Yaskawa INFORM job: TWIN_FRONT_WELD_-90ST-2_5340.JBI

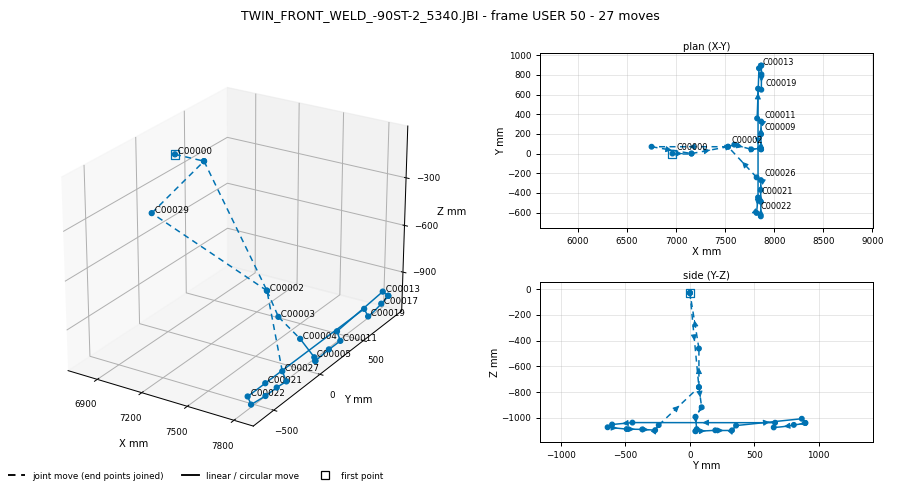
[picture p0: tool path of TWIN_FRONT_WELD_-90ST-2_5340.JBI in frame USER 50, 27 of 31 moves have a stored position in this frame; points joined in program order, loops and branches not executed]
/JOB
//NAME TWIN_FRONT_WELD_-90ST-2_5340
///FOLDERNAME 02-SKRZYNIE_JOBS
//POS
///NPOS 31,31,0,6,0,0
///USER 50
///TOOL 0
///POSTYPE USER
///RECTAN
///RCONF 0,0,1,0,0,0,0,0,0,0,0,0,0,0,0,0,0,0,0,0,0,0,0,0
C00000=6964.103,0.312,-30.113,0.0036,-53.6521,-0.0034
C00001=7158.107,0.312,-30.113,0.0036,-53.6521,-0.0034
///RCONF 1,0,0,0,0,0,0,0,0,0,0,0,0,0,0,0,0,0,0,0,0,0,0,0
C00002=7529.895,69.936,-761.128,0.1694,36.7808,-161.6994
C00003=7593.803,91.186,-917.296,-9.7230,35.0705,-163.2693
C00004=7765.973,43.237,-990.708,2.4332,41.3600,-160.2788
C00005=7854.092,52.836,-1087.295,2.4326,41.3464,-160.2685
C00006=7866.086,43.569,-1103.074,2.4250,41.3408,-160.2847
C00007=7866.672,43.652,-1103.070,2.4247,41.3414,-160.2846
C00008=7865.168,101.752,-1101.058,2.4312,41.5896,-160.2966
///RCONF 0,0,0,0,0,0,0,0,0,0,0,0,0,0,0,0,0,0,0,0,0,0,0,0
C00009=7865.744,197.178,-1096.159,2.5302,41.7008,-160.1737
C00010=7865.567,255.531,-1097.573,2.5319,41.6997,-160.1630
C00011=7866.686,326.732,-1096.309,2.5308,41.6996,-160.1597
C00012=7825.961,358.355,-1059.396,2.5279,41.7009,-160.1704
C00013=7844.512,868.318,-1006.408,-36.5717,33.3380,158.1479
C00014=7867.707,896.307,-1038.748,-33.3426,31.0834,153.4598
C00015=7867.746,895.180,-1038.953,-33.3375,31.0829,153.4546
C00016=7869.178,857.917,-1047.022,-33.1867,30.9856,153.2302
C00017=7869.794,806.472,-1054.108,-32.5616,29.0872,131.6988
C00018=7869.506,734.683,-1066.166,-32.5472,29.0702,136.7150
C00019=7868.451,650.382,-1073.764,-32.5333,29.0523,142.4520
C00020=7835.214,661.117,-1037.227,-32.5695,29.0775,153.4943
C00021=7835.222,-446.023,-1036.229,41.9938,34.9165,-143.3319
C00022=7820.199,-603.860,-1051.032,41.9928,34.9182,-143.3350
C00023=7863.342,-638.725,-1072.644,41.9898,34.9141,-143.3376
///RCONF 0,0,0,0,1,0,0,0,0,0,0,0,0,0,0,0,0,0,0,0,0,0,0,0
C00024=7863.688,-490.448,-1086.753,35.6266,29.1231,-116.2046
///RCONF 0,0,0,0,0,0,0,0,0,0,0,0,0,0,0,0,0,0,0,0,0,0,0,0
C00025=7862.301,-369.694,-1089.170,35.5308,29.0998,-115.5093
C00026=7864.181,-269.690,-1094.936,35.4517,29.0825,-114.8963
C00027=7820.806,-242.024,-1055.912,35.4344,29.0737,-114.7919
///RCONF 1,0,0,0,0,0,0,0,0,0,0,0,0,0,0,0,0,0,0,0,0,0,0,0
C00028=7529.895,69.936,-761.128,0.1694,36.7808,-161.6994
///RCONF 1,0,1,0,0,0,0,0,0,0,0,0,0,0,0,0,0,0,0,0,0,0,0,0
C00029=6751.458,69.938,-461.595,1.9967,40.9431,-160.5509
///RCONF 0,0,1,0,0,0,0,0,0,0,0,0,0,0,0,0,0,0,0,0,0,0,0,0
C00030=7158.107,0.312,-30.113,0.0036,-53.6521,-0.0034
///RCONF 0,0,0,0,0,0,0,0,0,0,0,0,0,0,0,0,0,0,0,0,0,0,0,0
BC00000=5149.685
BC00001=5343.689
BC00002=6178.800
BC00003=6423.804
BC00004=6624.475
BC00005=6624.475
BC00006=6624.495
BC00007=6624.495
BC00008=6624.488
BC00009=6624.482
BC00010=6624.482
BC00011=6624.482
BC00012=6624.482
BC00013=6624.488
BC00014=6624.488
BC00015=6624.488
BC00016=6624.476
BC00017=6624.489
BC00018=6624.489
BC00019=6624.228
BC00020=6624.488
BC00021=6624.488
BC00022=6624.482
BC00023=6624.482
BC00024=6624.469
BC00025=6624.475
BC00026=6624.482
BC00027=6624.482
BC00028=6178.800
BC00029=5343.689
BC00030=5343.689
///POSTYPE BASE
///RCONF 1,0,0,0,0,0,0,0,0,0,0,0,0,0,0,0,0,0,0,0,0,0,0,0
P00500=2.332,-5.281,-1.258,0.0000,0.0000,0.0000
///RCONF 0,0,0,0,0,0,0,0,0,0,0,0,0,0,0,0,0,0,0,0,0,0,0,0
P00501=-2.026,0.009,3.534,0.0000,0.0000,0.0000
///RCONF 1,0,0,0,0,0,0,0,0,0,0,0,0,0,0,0,0,0,0,0,0,0,0,0
P00502=-2.023,0.001,1.732,0.0000,0.0000,0.0000
P00503=0.138,-0.044,1.539,0.0000,0.0000,0.0000
P00504=-0.309,-0.010,1.636,0.0000,0.0000,0.0000
P00505=0.999,-9.916,8.214,0.0000,0.0000,0.0000
//INST
///DATE 2024/12/18 15:54
///ATTR SC,RW,RJ
////FRAME USER 50
///GROUP1 RB1,BS1
NOP
MOVJ C00000 BC00000 VJ=60.00
MOVJ C00001 BC00001 VJ=60.00
MOVJ C00002 BC00002 VJ=60.00
MOVJ C00003 BC00003 VJ=60.00
MOVJ C00004 BC00004 VJ=30.00
'::::::::::::::::::::::::::::::::
'W20
'::::::::::::::::::::::::::::::::
MOVL C00005 BC00005 V=333.3
SFTON P0503
MACRO1 MJ#(0) ARGF14
MOVL C00006 BC00006 V=166.7 PL=0
ARCON
MOVC C00007 BC00007 V=9.5
MOVC C00008 BC00008 V=9.5
MOVC C00009 BC00009 V=9.5
SFTOF
SFTON P0502
MOVC C00010 BC00010 V=9.5
MOVC C00011 BC00011 V=9.5
ARCOF
MOVL C00012 BC00012 V=166.7
SFTOF
'::::::::::::::::::::::::::::::::
'W21
'::::::::::::::::::::::::::::::::
MOVL C00013 BC00013 V=333.3
SFTON P0500
MACRO1 MJ#(0) ARGF14
MOVL C00014 BC00014 V=166.7 PL=0
ARCON
MOVC C00015 BC00015 V=9.5
MOVC C00016 BC00016 V=9.5
MOVC C00017 BC00017 V=9.5
SFTOF
SFTON P0501
MOVC C00018 BC00018 V=9.5
MOVC C00019 BC00019 V=9.5
ARCOF
MOVL C00020 BC00020 V=166.7
SFTOF
MOVL C00021 BC00021 V=333.3
'::::::::::::::::::::::::::::::::
'W22
'::::::::::::::::::::::::::::::::
MOVL C00022 BC00022 V=333.3
SFTON P0505
MACRO1 MJ#(0) ARGF14
MOVL C00023 BC00023 V=166.7 PL=0
ARCON
MOVL C00024 BC00024 V=10.0
SFTOF
SFTON P0504
MOVL C00025 BC00025 V=9.5
MOVL C00026 BC00026 V=10.0
ARCOF
MOVL C00027 BC00027 V=250.0
SFTOF
MOVJ C00028 BC00028 VJ=50.00
MOVJ C00029 BC00029 VJ=80.00
MOVJ C00030 BC00030 VJ=80.00
END
